(* Schneider Machine Expert - Basic project exercise_3.1, file version 2.9.0.0 *)
(* ProjectInformations: Name=Novo projeto *)

HARDWARE
  Cpu 0: TM221CE24R
  EthernetConfiguration: NetworkName=M221, IpAllocationMode=FixedAddress, IpAddress=0.0.0.0, SubnetMask=0.0.0.0
  SerialLineConfiguration: Baud=Baud19200, Parity=ParityEven, DataBits=DataBits8, StopBits=StopBits1, PhysicalMedium=PhysicalMediumRs485, TransmissionMode=TransmissionModeModbusRtu, SlaveId=1, Addressing=SlaveAddressing
  MastTask: UsePeriodScanMode=false, PeriodScan=100
  FastTask: Period=255
  CpuBehavior: StartingMode=StartAsPreviousState, AutoSaveRamOnEeprom=true, WatchdogPeriod=250

SYMBOLS  (address, symbol, comment, settings)
  %M0       SIG_IN_SEN_A_ATU
  %M1       SIG_IN_SEN_A_DESA
  %M2       SIG_IN_SEN_B_ATU
  %M3       SIG_IN_SEN_B_DESA
  %M4       SIG_IN_SEN_C_ATU
  %M5       SIG_IN_SEN_C_DESA
  %M6       SIG_IN_SEN_D_ATU
  %M7       SIG_IN_SEN_D_DESA
  %M20      SIG_OUT_FECHA_ATU_P1
  %M21      SIG_OUT_ABRE_ATU_P1
  %M22      SIG_OUT_LIGA_ATU_M1
  %M23      SIG_OUT_DESL_ATU_M1
  %M24      SIG_OUT_LIGA_ATU_M2
  %M25      SIG_OUT_DESL_ATU_M2
  %M26      SIG_OUT_LIGA_ALA_AL1
  %M27      SIG_OUT_DESL_ALA_AL1
  %M51      SIG_OUT_MOT1
  %M52      SIG_OUT_MOT2
  %M53      SIG_OUT_VALV_P
  %I0.0     IN_SEN_A_ATU
  %I0.1     IN_SEN_A_DESA
  %I0.2     IN_SEN_B_ATU
  %I0.3     IN_SEN_B_DESA
  %I0.4     IN_SEN_C_ATU
  %I0.5     IN_SEN_C_DESA
  %I0.6     IN_SEN_D_ATU
  %I0.7     IN_SEN_D_DESA
  %Q0.1     ATU_M1
  %Q0.2     ATU_M2
  %Q0.3     ATU_P1
  %Q0.5     ALAR_AL

POU Entradas
  (* SectionNumber=1 *)

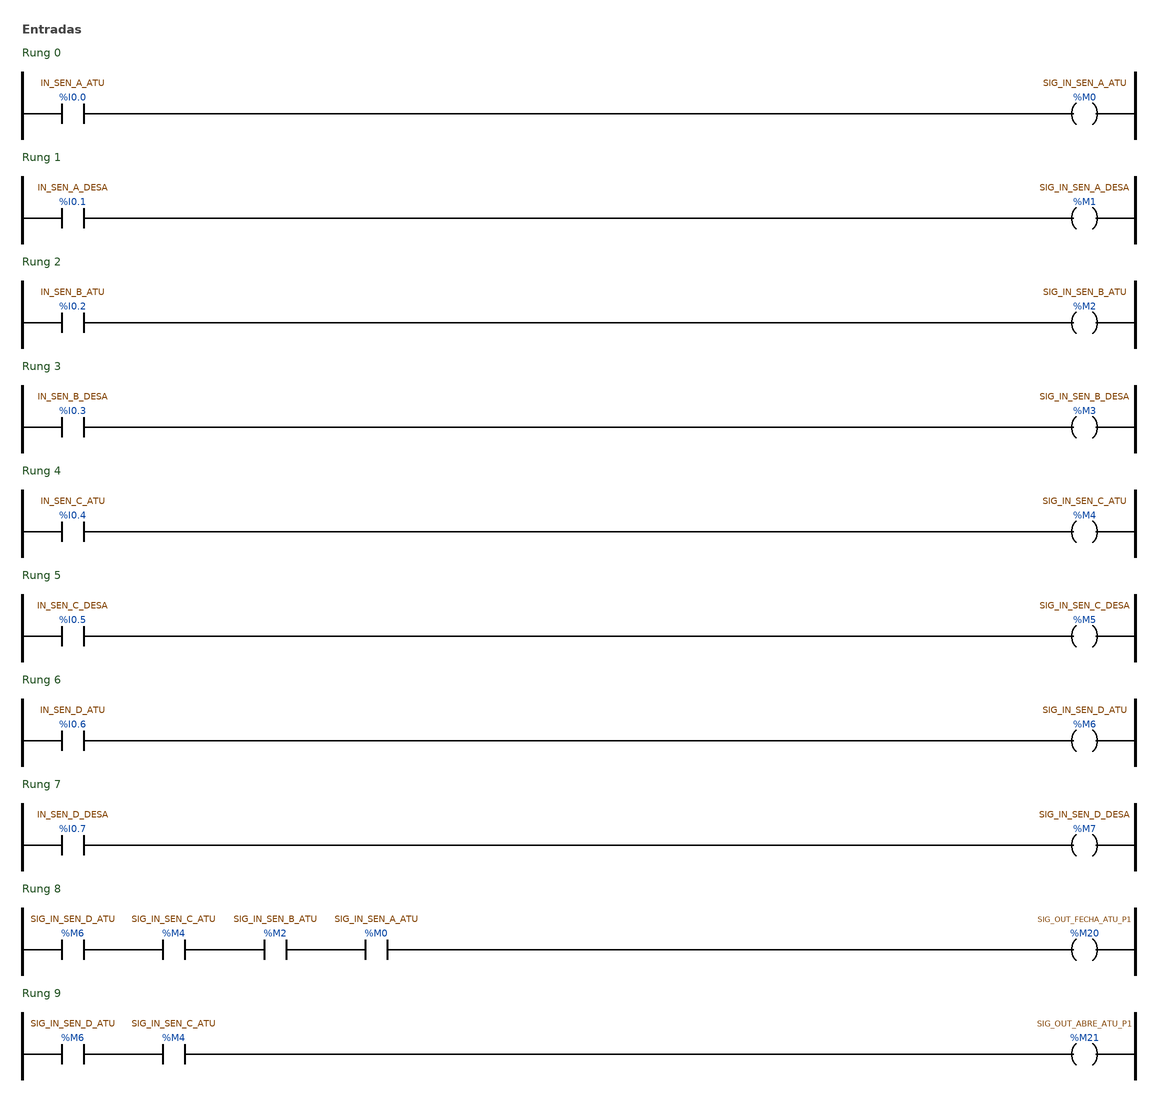

// Rung 0
  LD %I0.0                (* IN_SEN_A_ATU *)
  ST %M0                  (* SIG_IN_SEN_A_ATU *)
  // as ST:
  //   SIG_IN_SEN_A_ATU := IN_SEN_A_ATU;

// Rung 1
  LD %I0.1                (* IN_SEN_A_DESA *)
  ST %M1                  (* SIG_IN_SEN_A_DESA *)
  // as ST:
  //   SIG_IN_SEN_A_DESA := IN_SEN_A_DESA;

// Rung 2
  LD %I0.2                (* IN_SEN_B_ATU *)
  ST %M2                  (* SIG_IN_SEN_B_ATU *)
  // as ST:
  //   SIG_IN_SEN_B_ATU := IN_SEN_B_ATU;

// Rung 3
  LD %I0.3                (* IN_SEN_B_DESA *)
  ST %M3                  (* SIG_IN_SEN_B_DESA *)
  // as ST:
  //   SIG_IN_SEN_B_DESA := IN_SEN_B_DESA;

// Rung 4
  LD %I0.4                (* IN_SEN_C_ATU *)
  ST %M4                  (* SIG_IN_SEN_C_ATU *)
  // as ST:
  //   SIG_IN_SEN_C_ATU := IN_SEN_C_ATU;

// Rung 5
  LD %I0.5                (* IN_SEN_C_DESA *)
  ST %M5                  (* SIG_IN_SEN_C_DESA *)
  // as ST:
  //   SIG_IN_SEN_C_DESA := IN_SEN_C_DESA;

// Rung 6
  LD %I0.6                (* IN_SEN_D_ATU *)
  ST %M6                  (* SIG_IN_SEN_D_ATU *)
  // as ST:
  //   SIG_IN_SEN_D_ATU := IN_SEN_D_ATU;

// Rung 7
  LD %I0.7                (* IN_SEN_D_DESA *)
  ST %M7                  (* SIG_IN_SEN_D_DESA *)
  // as ST:
  //   SIG_IN_SEN_D_DESA := IN_SEN_D_DESA;

// Rung 8
  LD %M6                  (* SIG_IN_SEN_D_ATU *)
  AND %M4                 (* SIG_IN_SEN_C_ATU *)
  AND %M2                 (* SIG_IN_SEN_B_ATU *)
  AND %M0                 (* SIG_IN_SEN_A_ATU *)
  ST %M20                 (* SIG_OUT_FECHA_ATU_P1 *)
  // as ST:
  //   SIG_OUT_FECHA_ATU_P1 := SIG_IN_SEN_D_ATU AND SIG_IN_SEN_C_ATU AND SIG_IN_SEN_B_ATU AND SIG_IN_SEN_A_ATU;

// Rung 9
  LD %M6                  (* SIG_IN_SEN_D_ATU *)
  AND %M4                 (* SIG_IN_SEN_C_ATU *)
  ST %M21                 (* SIG_OUT_ABRE_ATU_P1 *)
  // as ST:
  //   SIG_OUT_ABRE_ATU_P1 := SIG_IN_SEN_D_ATU AND SIG_IN_SEN_C_ATU;

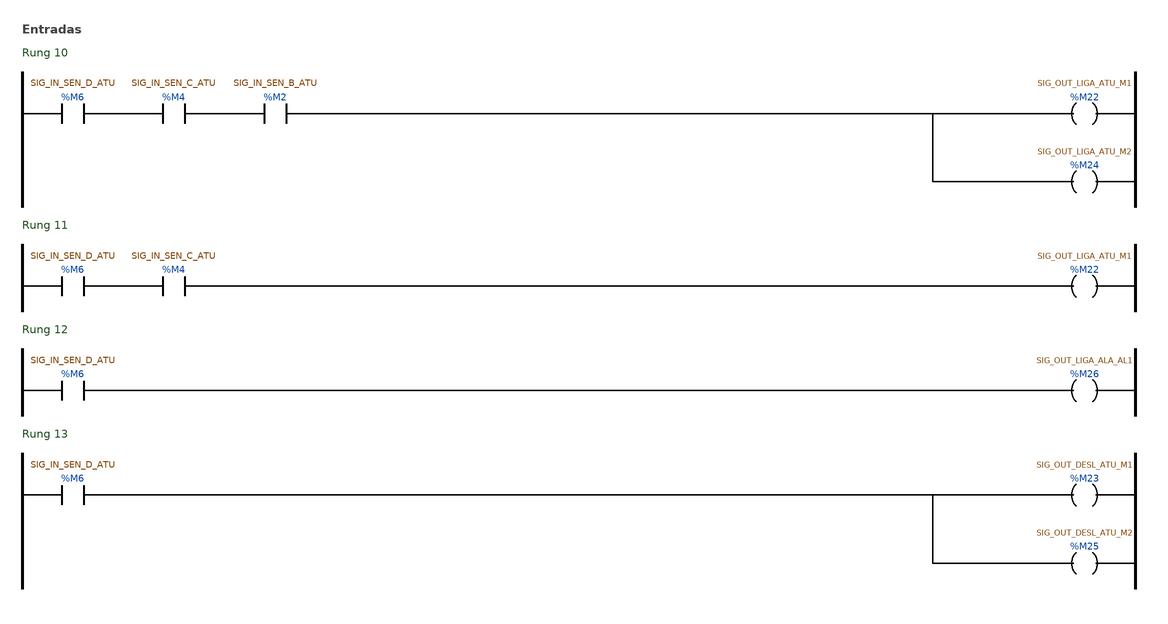

// Rung 10
  LD %M6                  (* SIG_IN_SEN_D_ATU *)
  AND %M4                 (* SIG_IN_SEN_C_ATU *)
  AND %M2                 (* SIG_IN_SEN_B_ATU *)
  ST %M22                 (* SIG_OUT_LIGA_ATU_M1 *)
  ST %M24                 (* SIG_OUT_LIGA_ATU_M2 *)
  // as ST:
  //   SIG_OUT_LIGA_ATU_M1 := SIG_IN_SEN_D_ATU AND SIG_IN_SEN_C_ATU AND SIG_IN_SEN_B_ATU;
  //   SIG_OUT_LIGA_ATU_M2 := SIG_IN_SEN_D_ATU AND SIG_IN_SEN_C_ATU AND SIG_IN_SEN_B_ATU;

// Rung 11
  LD %M6                  (* SIG_IN_SEN_D_ATU *)
  AND %M4                 (* SIG_IN_SEN_C_ATU *)
  ST %M22                 (* SIG_OUT_LIGA_ATU_M1 *)
  // as ST:
  //   SIG_OUT_LIGA_ATU_M1 := SIG_IN_SEN_D_ATU AND SIG_IN_SEN_C_ATU;

// Rung 12
  LD %M6                  (* SIG_IN_SEN_D_ATU *)
  ST %M26                 (* SIG_OUT_LIGA_ALA_AL1 *)
  // as ST:
  //   SIG_OUT_LIGA_ALA_AL1 := SIG_IN_SEN_D_ATU;

// Rung 13
  LD %M6                  (* SIG_IN_SEN_D_ATU *)
  ST %M23                 (* SIG_OUT_DESL_ATU_M1 *)
  ST %M25                 (* SIG_OUT_DESL_ATU_M2 *)
  // as ST:
  //   SIG_OUT_DESL_ATU_M1 := SIG_IN_SEN_D_ATU;
  //   SIG_OUT_DESL_ATU_M2 := SIG_IN_SEN_D_ATU;

POU Lógicas
  (* SectionNumber=2 *)

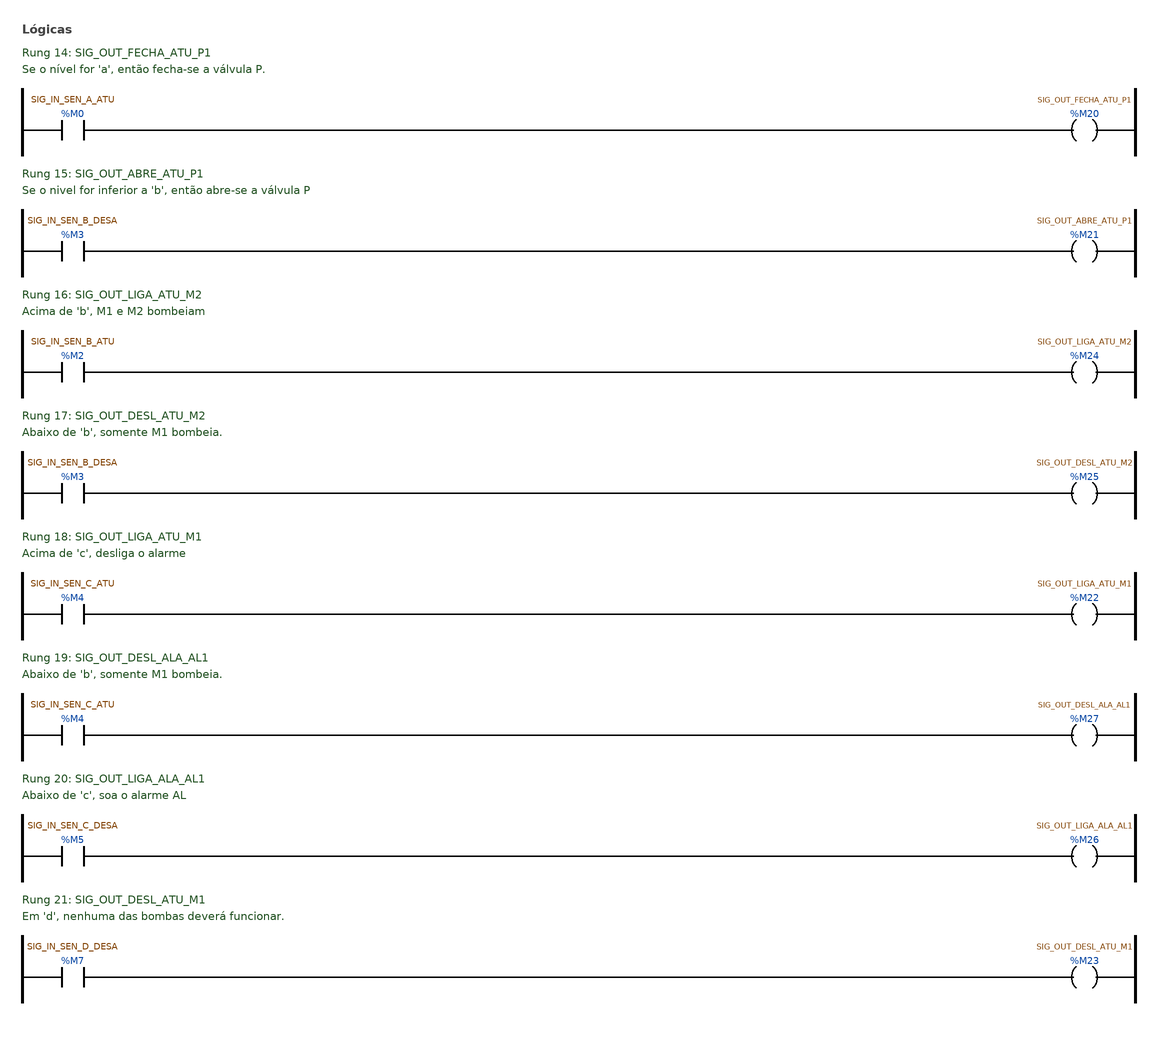

// Rung 14: SIG_OUT_FECHA_ATU_P1
// Se o nível for 'a', então fecha-se a válvula P.
  LD %M0                  (* SIG_IN_SEN_A_ATU *)
  ST %M20                 (* SIG_OUT_FECHA_ATU_P1 *)
  // as ST:
  //   SIG_OUT_FECHA_ATU_P1 := SIG_IN_SEN_A_ATU;

// Rung 15: SIG_OUT_ABRE_ATU_P1
// Se o nivel for inferior a 'b', então abre-se a válvula P
  LD %M3                  (* SIG_IN_SEN_B_DESA *)
  ST %M21                 (* SIG_OUT_ABRE_ATU_P1 *)
  // as ST:
  //   SIG_OUT_ABRE_ATU_P1 := SIG_IN_SEN_B_DESA;

// Rung 16: SIG_OUT_LIGA_ATU_M2
// Acima de 'b', M1 e M2 bombeiam
  LD %M2                  (* SIG_IN_SEN_B_ATU *)
  ST %M24                 (* SIG_OUT_LIGA_ATU_M2 *)
  // as ST:
  //   SIG_OUT_LIGA_ATU_M2 := SIG_IN_SEN_B_ATU;

// Rung 17: SIG_OUT_DESL_ATU_M2
// Abaixo de 'b', somente M1 bombeia.
  LD %M3                  (* SIG_IN_SEN_B_DESA *)
  ST %M25                 (* SIG_OUT_DESL_ATU_M2 *)
  // as ST:
  //   SIG_OUT_DESL_ATU_M2 := SIG_IN_SEN_B_DESA;

// Rung 18: SIG_OUT_LIGA_ATU_M1
// Acima de 'c', desliga o alarme
  LD %M4                  (* SIG_IN_SEN_C_ATU *)
  ST %M22                 (* SIG_OUT_LIGA_ATU_M1 *)
  // as ST:
  //   SIG_OUT_LIGA_ATU_M1 := SIG_IN_SEN_C_ATU;

// Rung 19: SIG_OUT_DESL_ALA_AL1
// Abaixo de 'b', somente M1 bombeia.
  LD %M4                  (* SIG_IN_SEN_C_ATU *)
  ST %M27                 (* SIG_OUT_DESL_ALA_AL1 *)
  // as ST:
  //   SIG_OUT_DESL_ALA_AL1 := SIG_IN_SEN_C_ATU;

// Rung 20: SIG_OUT_LIGA_ALA_AL1
// Abaixo de 'c', soa o alarme AL
  LD %M5                  (* SIG_IN_SEN_C_DESA *)
  ST %M26                 (* SIG_OUT_LIGA_ALA_AL1 *)
  // as ST:
  //   SIG_OUT_LIGA_ALA_AL1 := SIG_IN_SEN_C_DESA;

// Rung 21: SIG_OUT_DESL_ATU_M1
// Em 'd', nenhuma das bombas deverá funcionar.
  LD %M7                  (* SIG_IN_SEN_D_DESA *)
  ST %M23                 (* SIG_OUT_DESL_ATU_M1 *)
  // as ST:
  //   SIG_OUT_DESL_ATU_M1 := SIG_IN_SEN_D_DESA;

POU Saídas
  (* SectionNumber=3 *)

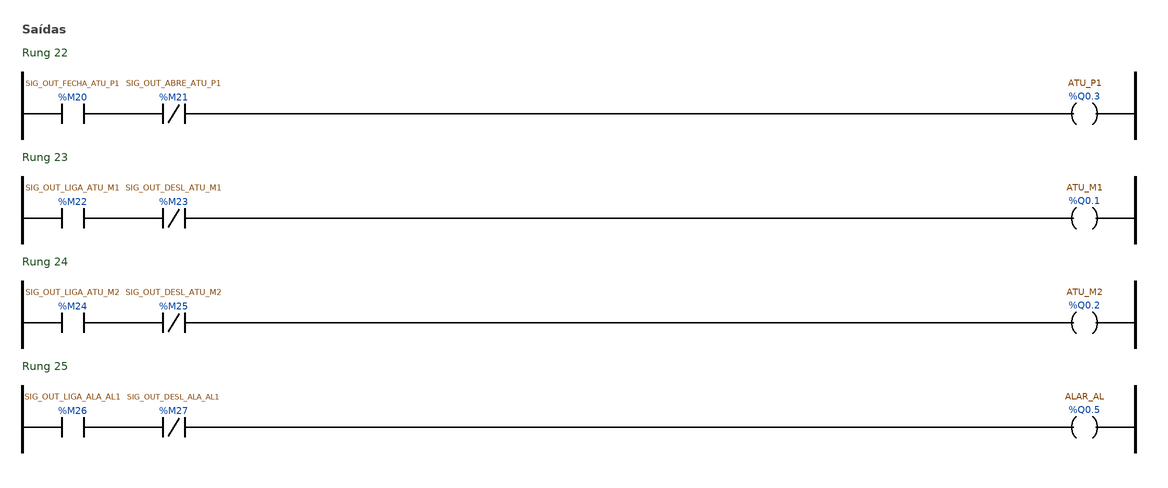

// Rung 22
  LD %M20                 (* SIG_OUT_FECHA_ATU_P1 *)
  ANDN %M21               (* SIG_OUT_ABRE_ATU_P1 *)
  ST %Q0.3                (* ATU_P1 *)
  // as ST:
  //   ATU_P1 := SIG_OUT_FECHA_ATU_P1 AND NOT SIG_OUT_ABRE_ATU_P1;

// Rung 23
  LD %M22                 (* SIG_OUT_LIGA_ATU_M1 *)
  ANDN %M23               (* SIG_OUT_DESL_ATU_M1 *)
  ST %Q0.1                (* ATU_M1 *)
  // as ST:
  //   ATU_M1 := SIG_OUT_LIGA_ATU_M1 AND NOT SIG_OUT_DESL_ATU_M1;

// Rung 24
  LD %M24                 (* SIG_OUT_LIGA_ATU_M2 *)
  ANDN %M25               (* SIG_OUT_DESL_ATU_M2 *)
  ST %Q0.2                (* ATU_M2 *)
  // as ST:
  //   ATU_M2 := SIG_OUT_LIGA_ATU_M2 AND NOT SIG_OUT_DESL_ATU_M2;

// Rung 25
  LD %M26                 (* SIG_OUT_LIGA_ALA_AL1 *)
  ANDN %M27               (* SIG_OUT_DESL_ALA_AL1 *)
  ST %Q0.5                (* ALAR_AL *)
  // as ST:
  //   ALAR_AL := SIG_OUT_LIGA_ALA_AL1 AND NOT SIG_OUT_DESL_ALA_AL1;
